% RSLogix 500 project 10.1.RSS, saved by version 8.30.00.16 %
PROJECT "10"    % processor: Bul.1763 MicroLogix 1100 Series B %

PROGRAM FILES
  LAD 2   4 rungs

DATA FILES
  O0 OUTPUT  4 elements
  I1 INPUT  6 elements
  S2 STATUS  66 elements
  B3 BINARY  1 elements
  T4 TIMER  1 elements
  C5 COUNTER  1 elements
  R6 CONTROL  1 elements
  N7 INTEGER  5 elements
  F8 FLOAT  1 elements

LADDER 2
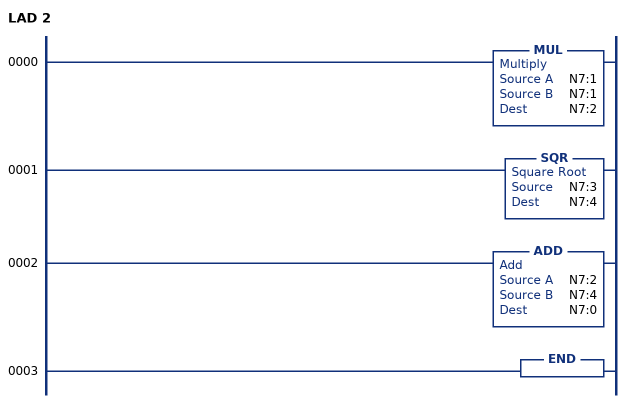
% Rung: 0 %
SOR MUL N7:1 N7:1 N7:2 EOR
% Rung: 1 %
SOR SQR N7:3 N7:4 EOR
% Rung: 2 %
SOR ADD N7:2 N7:4 N7:0 EOR
% Rung: 3 %
SOR END EOR
